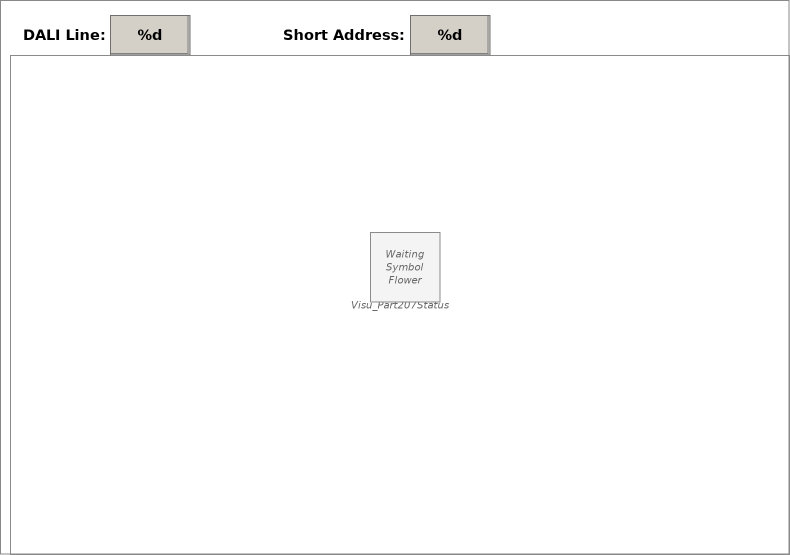
VISUALIZATION Visu_Part207  // 790x555
    Group (280,15 210x40)
        Textfield (0,0 130x40), "Short Address:"
        Button (130,0 80x40), "%d", text variable: DALI_Commissioning.fbPart207LED.nAddress
            OnMouseClick: write the text variable via Default, min 0, max 63, title "Insert Short Address"
    Group (20,15 170x40)
        Textfield (0,0 110x40), "DALI Line:"
        Button (90,0 80x40), "%d", text variable: GVL_Internal.nDALILine
            OnMouseClick: write the text variable via Default, min 1, max 10, title "Choose line"
    TabControl (10,55 780x500)
        shows Visu_Part207Status()
        shows Visu_Part207Parameters()
        shows Test()
        [0]: TabTitle=Status LED
        [1]: TabTitle=Parameters LED
        [2]: TabTitle=Paremeters LED
    WaitingSymbolFlower (370,232 70x70), invisible if: DALI_Commissioning.fbPart207LED.bHideWaitSymbol
END_VISUALIZATION

(* stored: Version 1.1.0.1
   Visu Visu_Part207: Id {ad2435a7-285f-4b30-8833-661a8d715c6b} *)
